(* Base of Control Primitives. Inheriting FBs must implement the type-specific "ExecuteInternal" method. *)
FUNCTION_BLOCK ABSTRACT ControlPrimitiveBase EXTENDS BehaviorBase
VAR
	m_timeout: TIME;
	
	m_internalRes: BOOL;
	m_pre: IExpression;
	m_post: IExpression;
	
	// store the conditions as string for access via OPC UA + easier debugging
	m_preStr: STRING(256);
	m_postStr: STRING(256);
	
	m_st: POINTER TO StateTracker;
	m_ra: POINTER TO RaConnector;
	
	m_tonTimeout: TON;
	
	m_didAbort: BOOL;
END_VAR

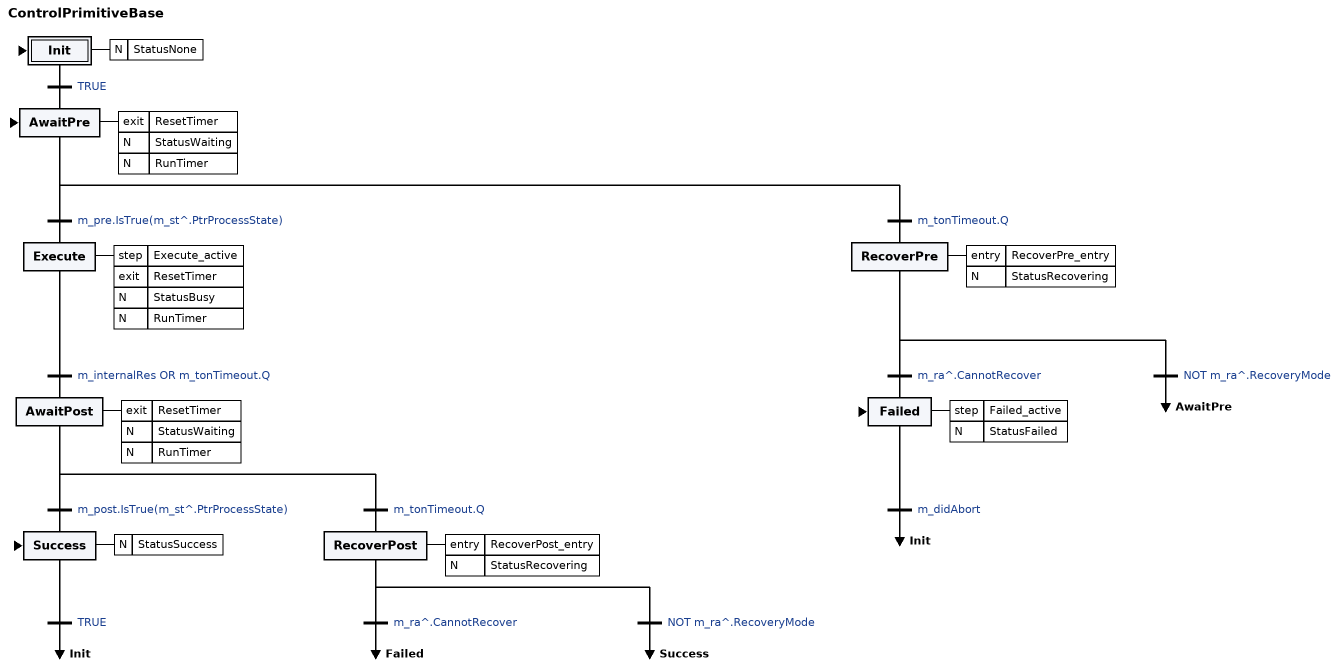
INITIAL_STEP Init:
    StatusNone(N);
END_STEP
TRANSITION FROM Init TO AwaitPre
    := TRUE;
END_TRANSITION
STEP AwaitPre:
    ResetTimer(P0);  // exit action
    StatusWaiting(N);
    RunTimer(N);
END_STEP
TRANSITION FROM AwaitPre TO Execute
    := m_pre.IsTrue(m_st^.PtrProcessState);
END_TRANSITION
STEP Execute:
    Execute_active(N);  // step action
    ResetTimer(P0);  // exit action
    StatusBusy(N);
    RunTimer(N);
END_STEP
TRANSITION FROM Execute TO AwaitPost
    := m_internalRes OR m_tonTimeout.Q;
END_TRANSITION
STEP AwaitPost:
    ResetTimer(P0);  // exit action
    StatusWaiting(N);
    RunTimer(N);
END_STEP
TRANSITION FROM AwaitPost TO Success
    := m_post.IsTrue(m_st^.PtrProcessState);
END_TRANSITION
STEP Success:
    StatusSuccess(N);
END_STEP
TRANSITION FROM Success TO Init
    := TRUE;
END_TRANSITION
TRANSITION FROM AwaitPost TO RecoverPost
    := m_tonTimeout.Q;
END_TRANSITION
STEP RecoverPost:
    RecoverPost_entry(P1);  // entry action
    StatusRecovering(N);
END_STEP
TRANSITION FROM RecoverPost TO Failed
    := m_ra^.CannotRecover;
END_TRANSITION
TRANSITION FROM RecoverPost TO Success
    := NOT m_ra^.RecoveryMode;
END_TRANSITION
TRANSITION FROM AwaitPre TO RecoverPre
    := m_tonTimeout.Q;
END_TRANSITION
STEP RecoverPre:
    RecoverPre_entry(P1);  // entry action
    StatusRecovering(N);
END_STEP
TRANSITION FROM RecoverPre TO Failed
    := m_ra^.CannotRecover;
END_TRANSITION
STEP Failed:
    Failed_active(N);  // step action
    StatusFailed(N);
END_STEP
TRANSITION FROM Failed TO Init
    := m_didAbort;
END_TRANSITION
TRANSITION FROM RecoverPre TO AwaitPre
    := NOT m_ra^.RecoveryMode;
END_TRANSITION

METHOD Abort : BOOL
VAR_INPUT
END_VAR
END_METHOD

ACTION Execute_active:
IF NOT m_internalRes THEN
	m_internalRes := ExecuteInternal(i_params);
END_IF
END_ACTION

(* Execution logic of this Control Primitive. *)
METHOD PROTECTED ABSTRACT ExecuteInternal : BOOL
VAR_INPUT
	i_params: ParameterSet;
END_VAR
END_METHOD

ACTION Failed_active:
m_didAbort := Abort();
END_ACTION

PROPERTY Postcondition : IExpression
GET
Postcondition := m_post;
END_GET
SET
m_post := Postcondition;
m_postStr := Postcondition.ToString();
END_SET
END_PROPERTY

PROPERTY Precondition : IExpression
GET
Precondition := m_pre;
END_GET
SET
m_pre := Precondition;
m_preStr := Precondition.ToString();
END_SET
END_PROPERTY

METHOD ProvideServices : BOOL
VAR_INPUT
	i_ptrRaConnector: POINTER TO RaConnector;
	i_ptrStateTracker: POINTER TO StateTracker;
END_VAR
m_ra := i_ptrRaConnector;
m_st := i_ptrStateTracker;
END_METHOD

ACTION RecoverPost_entry:
m_ra^.RequestRecovery(m_post, CONCAT('Primitive ', TO_STRING(m_id)));
END_ACTION

ACTION RecoverPre_entry:
m_ra^.RequestRecovery(m_pre, CONCAT('Primitive ', TO_STRING(m_id)));
END_ACTION

ACTION ResetTimer:
m_tonTimeout(IN := FALSE);
m_internalRes := FALSE;
END_ACTION

ACTION RunTimer:
m_tonTimeout(IN := TRUE, PT := m_timeout);
END_ACTION

ACTION StatusBusy:
o_status := EOperationResult.busy;
END_ACTION

ACTION StatusFailed:
o_status := EOperationResult.failed;
END_ACTION

ACTION StatusNone:
o_status := EOperationResult.none;
END_ACTION

ACTION StatusRecovering:
o_status := EOperationResult.recovering;
END_ACTION

ACTION StatusSuccess:
o_status := EOperationResult.success;
END_ACTION

ACTION StatusWaiting:
o_status := EOperationResult.waiting;
END_ACTION

END_FUNCTION_BLOCK

(* stored: Version 1.1.0.1, ProductVersion 3.1.4024.12
   POU ControlPrimitiveBase: Id {7ed5e3b2-8b7a-496e-8688-2a61da6a4089}, SpecialFunc None
   Folder Actions: Id {62a85686-4f23-4c67-b676-ab492ae41d1d}
   Method Abort: Id {d9bf888c-380c-4202-bf03-1e27f2b8b9ed}
   Action Execute_active: Id {88921597-abf9-4360-b60c-9c68454ab9a0}
   Method ExecuteInternal: Id {c276dbfb-d3fb-4c4b-b87f-50ae91f391d6}
   Action Failed_active: Id {ffaa7d8d-1e5c-4b08-b199-cecd33b8a5c8}
   Property Postcondition: Id {551dc54f-bfd8-47cc-ba12-6deb36a4dee7}
   Get Get: Id {f04392f3-4a98-4642-9c8b-c7cfc146fd49}
   Set Set: Id {09c3e89e-62d3-492a-8438-4648a23ceb5e}
   Property Precondition: Id {c40e6ae4-ebc8-419c-b929-1938cfea6323}
   Get Get: Id {304a8eb1-2874-4141-a47b-e5579b51cc75}
   Set Set: Id {0734878d-df85-4026-919e-23988703e28c}
   Method ProvideServices: Id {9acd35f1-157a-4c50-a365-66d1f8a6daa7}
   Action RecoverPost_entry: Id {ea2cbcd9-e1e5-4cef-b31b-a8ab328b1151}
   Action RecoverPre_entry: Id {f638059f-27d1-40ab-bf8d-2585fb0204cc}
   Action ResetTimer: Id {77b33412-9ed7-495d-9c9f-c497e5485552}
   Action RunTimer: Id {9ddaccaf-8828-4c45-818a-670a2a751989}
   Action StatusBusy: Id {5be5c250-8cbd-4faa-9c04-d3e155956939}
   Action StatusFailed: Id {94861b87-5893-4eda-bd58-89ec69baf500}
   Action StatusNone: Id {41661edc-7a9e-45a5-a69a-c880702e7474}
   Action StatusRecovering: Id {944578b7-6909-43ec-9240-becb4c3c2065}
   Action StatusSuccess: Id {b1e98722-b6c8-42d4-aab3-10dba99a0e80}
   Action StatusWaiting: Id {ebcebbca-0086-4acc-932a-59a4327a92a8} *)
